(* IEC 61131-3 sources: AXOpen/src/templates.simple/ctrl/src/SampleControlledUnit, 6 files *)

(* ---- AutomatSequence.st ---- *)
USING AXOpen.Core;

NAMESPACE axosimple.SampleControlledUnit
    {#ix-set:AttributeName = "<#AUTOMAT#>"}
    CLASS PUBLIC AutomatSequence EXTENDS AXOpen.Core.AxoSequencer
        VAR PUBLIC
            Steps : ARRAY[0..150] OF AxoStep;
        END_VAR

        METHOD PUBLIC Run
            VAR_INPUT
                parent : IAxoObject;
            END_VAR
            VAR_IN_OUT
                Components : Components;
            END_VAR

            THIS.Initialize(parent);
            THIS.SequenceMode := eAxoSequenceMode#Cyclic;

            THIS.Open();
            THIS.AndThen(Steps[0],components.VerticalCylinder.MoveToWork);
            THIS.AndThen(Steps[1],components.GripperCylinder.MoveToWork);
            THIS.AndThen(Steps[2],components.VerticalCylinder.MoveToHome);
            THIS.AndThen(Steps[3],components.HorizontalCylinder.MoveToWork);
            THIS.AndThen(Steps[4],components.VerticalCylinder.MoveToWork);
            THIS.AndThen(Steps[5],components.GripperCylinder.MoveToHome);
            THIS.AndThen(Steps[6],components.VerticalCylinder.MoveToHome);
            THIS.AndThen(Steps[7],components.HorizontalCylinder.MoveToHome);
            THIS.AndThen(Steps[8],components.GripperCylinder.MoveToHome);
            THIS.Close(Steps[150]);

        END_METHOD
    END_CLASS
END_NAMESPACE

(* ---- Components.st ---- *)
USING AXOpen.Core;

NAMESPACE axosimple.SampleControlledUnit
    CLASS Components EXTENDS AXOpen.Core.AxoObject
        VAR PUBLIC
            HorizontalCylinder : AXOpen.Pneumatics.Cylinder;
            VerticalCylinder : AXOpen.Pneumatics.Cylinder;
            GripperCylinder : AXOpen.Pneumatics.Cylinder;
        END_VAR
        METHOD PUBLIC Update
            VAR_INPUT
                parent : IAxoObject;
            END_VAR
            VAR_IN_OUT
                Inputs : axosimple.Inputs;
                Outputs : axosimple.Outputs;
            END_VAR
            THIS.Initialize(parent);
            HorizontalCylinder.Update(THIS,Inputs.B0[0], Inputs.B0[1], Outputs.B0[0], Outputs.B0[1]);
            VerticalCylinder.Update(THIS,Inputs.B0[2], Inputs.B0[3], Outputs.B0[2], Outputs.B0[3]);
            GripperCylinder.Update(THIS,Inputs.B0[4], Inputs.B0[5], Outputs.B0[4], Outputs.B0[5]);
        END_METHOD
    END_CLASS

END_NAMESPACE

(* ---- ControlledUnit.st ---- *)
USING AXOpen.Core;

NAMESPACE axosimple.SampleControlledUnit
    CLASS ControlledUnit EXTENDS AXOpen.Core.AxoObject
        VAR PUBLIC
            GroundSequence : GroundSequence;
            AutomatSequence : AutomatSequence;
            ServiceMode : ServiceMode;
            Components : Components;
        END_VAR

        METHOD PUBLIC Run
            VAR_INPUT
                parent : IAxoContext;
            END_VAR
            VAR_IN_OUT
                Inputs : axosimple.Inputs;
                Outputs : axosimple.Outputs;
            END_VAR
            THIS.Initialize(parent);
            THIS.Execute(Inputs, Outputs);
        END_METHOD

        METHOD PUBLIC Run
            VAR_INPUT
                parent : IAxoObject;
            END_VAR
            VAR_IN_OUT
                Inputs : axosimple.Inputs;
                Outputs : axosimple.Outputs;
            END_VAR
            THIS.Initialize(parent);
            THIS.Execute(Inputs, Outputs);
        END_METHOD

        METHOD PRIVATE Execute
            VAR_IN_OUT
                Inputs : axosimple.Inputs;
                Outputs : axosimple.Outputs;
            END_VAR

            Components.Update(THIS,Inputs, Outputs);

            GroundSequence.Run(THIS, Components);

            IF(GroundSequence.IsBusy()) THEN
                AutomatSequence.Restore();
                ServiceMode.Restore();
            END_IF;

            AutomatSequence.IsDisabled := GroundSequence.Status <> eAxoTaskState#Done;
            AutomatSequence.Run(THIS, Components);

            ServiceMode.Run(THIS, Components);
            IF ServiceMode.IsBusy() THEN
                GroundSequence.Restore();
            END_IF;
        END_METHOD

    END_CLASS
END_NAMESPACE

(* ---- GroundSequence.st ---- *)
USING AXOpen.Core;

NAMESPACE axosimple.SampleControlledUnit
    {#ix-set:AttributeName = "<#GROUND#>"}
    CLASS PUBLIC GroundSequence EXTENDS AXOpen.Core.AxoSequencer
        VAR PUBLIC
            Steps : ARRAY[0..20] OF AxoStep;
        END_VAR

        METHOD PUBLIC Run
            VAR_INPUT
                parent : IAxoObject;
            END_VAR
            VAR_IN_OUT
                components : Components;
            END_VAR

            THIS.Initialize(parent);
            THIS.SequenceMode := eAxoSequenceMode#RunOnce;

            THIS.Open();
            THIS.AndThen(Steps[0],components.VerticalCylinder.MoveToHome);
            THIS.AndThen(Steps[1],components.HorizontalCylinder.MoveToHome);
            THIS.AndThen(Steps[2],components.GripperCylinder.MoveToHome);
            THIS.Close(Steps[3]);

        END_METHOD
    END_CLASS
END_NAMESPACE

(* ---- ProcessData.st ---- *)
USING AXOpen.Core;

NAMESPACE axosimple.SampleControlledUnit
    CLASS ProcessData
        VAR PUBLIC

        END_VAR
    END_CLASS
END_NAMESPACE

(* ---- ServiceMode.st ---- *)
USING AXOpen.Core;

NAMESPACE axosimple.SampleControlledUnit
    {#ix-set:AttributeName = "<#SERVICE#>"}
    CLASS PUBLIC ServiceMode EXTENDS AXOpen.Core.AxoTask
        METHOD PUBLIC Run
            VAR_INPUT
                parent : IAxoObject;
            END_VAR
            VAR_IN_OUT
                components : Components;
            END_VAR

            THIS.Initialize(parent);

            IF THIS.Execute() THEN
                THIS.Handle(components);
            END_IF;
        END_METHOD

        METHOD PRIVATE Handle
            VAR_IN_OUT
                components : Components;
            END_VAR
            components.HorizontalCylinder.ActivateManualControl();
            components.VerticalCylinder.ActivateManualControl();
            components.GripperCylinder.ActivateManualControl();
        END_METHOD

    END_CLASS
END_NAMESPACE
